// Mitsubishi GX Works2 project: z01   PLC: Q02/Q02H

PROGRAM MAIN
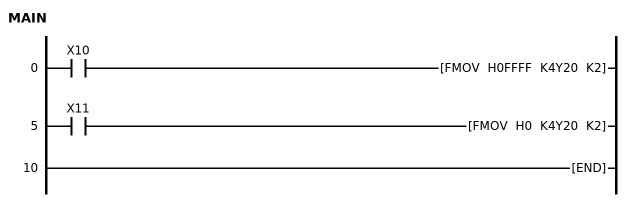
0     LD      X10
      FMOV    H0FFFF K4Y20 K2
5     LD      X11
      FMOV    H0 K4Y20 K2
10    END
END_PROGRAM
